{attribute 'qualified_only'}
{attribute 'strict'}
{attribute 'to_string'}
TYPE c3LnSwFaultCodes :
(
	InvalidTrafficControl := 0,
	InvalidOutputLane := 1
);
END_TYPE

(* stored: Version 1.1.0.1, ProductVersion 3.1.4024.6
   DUT c3LnSwFaultCodes: Id {fd4afb6d-28dc-4ced-860a-4acb33be1e7f} *)
